PROGRAM PressureControl
//VAR
//	iPressureScaledValue: INT; //Scaled pressure value
//	sFillingValveState: STRING; // Filling valve state in str
//	fillingValveAutoMode: BOOL;
//	sFillingValveControlState: STRING;
//	toggleFillingValve : FB_ToggleHeartBeat;
//	fTrigFillingAutoMode: F_TRIG;
//	rTrigFillingAutoMode: R_TRIG;
//	ReactorPressurePIDcontrol: FB_PIDsetpointOutput;
//	tonPressureControl: TON;
	
//	// PID params
//	PB: REAL :=7;
//	Ti: REAL := 10;
//	Td: REAL := 1;
//	Kp: REAL := 100/PB;
//	Ki: REAL := 1/Ti;
//	Kd: REAL := 1/Td;
//	PressureTestValue: REAL;
//	togglePressureControl: FB_ToggleHeartBeat;
//	ReactorPressureAutoPID : BOOL;
//	reactorPressureSetpoint: REAL;
//END_VAR
//VAR PERSISTENT
////	fillingValveOpenInterval: INT;
////	fillingValveCloseInterval: INT;	
//END_VAR

// Scale analog pressure
//iPressureScaledValue := F_AnalogScale(AnalogInputRawValue := IO.reactorPressure, MaxAnalogValue := 1000);
//// Manual operation of filling valve: state texts
//IF NOT io.reactorInletValve THEN
//	sFillingValveState := 'OPEN';
//ELSE
//	sFillingValveState := 'CLOSE';
//END_IF

//// Filling valve control mode and auto control
//IF fillingValveAutoMode THEN
//	sFillingValveControlState := 'AUTO';
//	toggleFillingValve(I_OpenInterValSecs := fillingValveOpenInterval, I_CloseIntervalSecs := fillingValveCloseInterval, O_Update => io.reactorInletValve);
//ELSE
//	sFillingValveControlState := 'MAN';
//END_IF
//// Open valve when auto mode is entered
//rTrigFillingAutoMode(CLK := fillingValveAutoMode);
//IF rTrigFillingAutoMode.Q THEN
//	//toggleFillingValve.firstTime(entered := TRUE);
//	io.reactorInletValve := TRUE;
//END_IF
//// Close valve when auto mode is entered
//fTrigFillingAutoMode(CLK := fillingValveAutoMode);
//IF fTrigFillingAutoMode.Q THEN
//	io.reactorInletValve := FALSE;
//END_IF


//(*togglePressureControl(I_OpenInterValSecs:= 1,
//					I_CloseIntervalSecs := ,
//					)*)
//IF ReactorPressureAutoPID THEN
//	ReactorPressurePIDcontrol(
//		Kp:= Kp, 
//		Ki:= Ki, 
//		Kd:= Kd, 
//		Bias:=0 , 
//		processVariable:= iPressureScaledValue,//PressureTestValue,
//		setpoint:= reactorPressureSetpoint, 
//		PIDy=> );
//ELSE
//	ReactorPressurePIDcontrol.ResetValues(TRUE);
//END_IF

//// PRESSURE PID CONTROL

END_PROGRAM

(* stored: Version 1.1.0.1, ProductVersion 3.1.4024.9
   POU PressureControl: Id {af9f6ef1-62a5-4326-9fa7-845cc278eb15}, SpecialFunc None *)
